VAR
	Document	  : SJsonValue;
	JsonAttribute : T_MaxString;
	TaskName	  : T_MaxString;
	temp		  : UDINT;
END_VAR

VAR_INST
	LastScanCount		 : UDINT;
	MessagesSentThisScan : UDINT;
	MissedMessages		 : UDINT;
	Throttled			 : BOOL;
END_VAR

VAR
	ThrottledNotificationString : T_MaxString;
	CurrentDCTime				: DCTIMESTRUCT;
	DCTime100Nsec				: WORD;
	DCTimeString				: T_MaxString;
END_VAR
IF NOT InitComplete THEN
	RETURN;
END_IF

{analysis -62}
IF NOT TracingAllowed THEN
	RETURN;
END_IF

IF NOT Parameters_Tracing.ALLOW_DUPLICATE_SEQUENTIAL_MESSAGES THEN
	IF (MEMCMP(ADR(Source), ADR(Previous_AddEntryJsonSource), SIZEOF(T_MaxString)) = 0) AND (MEMCMP(ADR(Message), ADR(Previous_AddEntryJsonMessage), SIZEOF(T_MaxString)) = 0) AND (Flags = Previous_AddEntryJsonFlags) AND (MEMCMP(ADR(Json), ADR(Previous_AddEntryJson), SIZEOF(T_MaxString)) = 0) THEN
		// This message is identical to the last message sent--ignore
		RETURN;
	END_IF
END_IF

Event.ipArguments.Clear().AddString(Message);
AddContext(Source := Source, Flags := Flags);
Document := JsonParser.NewDocument();
JsonParser.AddJsonMember(Document, 'ExtendedInfo', Json);
JsonAttribute := JsonParser.GetJson(Document);
Event.SetJsonAttribute(JsonAttribute);
Event.Send(0);
MessagesSentThisScan := MessagesSentThisScan + 1;
MEMCPY(ADR(Previous_AddEntryJsonSource), ADR(Source), SIZEOF(T_MaxString));
MEMCPY(ADR(Previous_AddEntryJsonMessage), ADR(Message), SIZEOF(T_MaxString));
Previous_AddEntryFlags := Flags;
MEMCPY(ADR(Previous_AddEntryJsonMessage), ADR(Json), SIZEOF(T_MaxString));
END_METHOD

METHOD FB_init : BOOL
VAR_INPUT
	bInitRetains : BOOL; // if TRUE, the retain variables are initialized (warm start / cold start)
	bInCopyCode	 : BOOL; // if TRUE, the instance afterwards gets moved into the copy code (online change)
END_VAR

VAR
	hr : HRESULT;
END_VAR
{analysis -15}
IF NOT Event.EqualsToEventEntryEx(TC_EVENTS.Tracing.TraceEvent) THEN
	IF SUCCEEDED(Event.CreateEx(TC_EVENTS.Tracing.TraceEvent, 0)) THEN
		InitComplete := TRUE;
	END_IF
ELSE
	InitComplete := TRUE;
END_IF
END_METHOD

PROPERTY PRIVATE TracingAllowed : BOOL
GET
VAR_INST
	LastScanCount  : UDINT;
	MissedMessages : UDINT;
	Throttled	   : BOOL;
END_VAR

VAR
	ThrottledNotificationString : T_MaxString;
END_VAR
{analysis -62}
IF NOT Parameters_Tracing.TRACING_ENABLED THEN
	TracingAllowed := FALSE;
	RETURN;
END_IF

IF TwinCAT_SystemInfoVarList._TaskInfo[GETCURTASKINDEXEX()].CycleCount = LastScanCount THEN
	// Trying to send multiple messages in same scan
	IF Throttled THEN
		MissedMessages := MissedMessages + 1;
		RETURN;
	ELSIF MessagesSentThisScan >= Parameters_Tracing.MAX_LOG_ENTRIES_PER_SCAN AND NOT Throttled THEN
		// Need to throttle messsage queue
		Event.ipArguments.Clear().AddString('Too many messages sent in single scan; tracing throttled.');
		Event.Send(0);
		MissedMessages := MissedMessages + 1;
		Throttled	   := TRUE;
		TracingAllowed := FALSE;
		RETURN;
	ELSE
		TracingAllowed := TRUE;
	END_IF
ELSE
	IF Throttled THEN
		ThrottledNotificationString := CONCAT('Missed ', CONCAT(TO_STRING(MissedMessages), ' throttled messages previously.'));
		Event.ipArguments.Clear().AddString(ThrottledNotificationString);
		Event.Send(0);
		MissedMessages := 0;
	END_IF

	LastScanCount		 := TwinCAT_SystemInfoVarList._TaskInfo[GETCURTASKINDEXEX()].CycleCount;
	MessagesSentThisScan := 0;
	Throttled			 := FALSE;
	TracingAllowed		 := TRUE;
END_IF
END_GET
END_PROPERTY

END_FUNCTION_BLOCK

// VISUs/V_MachineModule
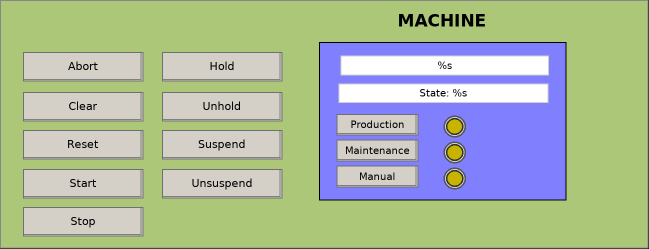
VISUALIZATION V_MachineModule  // 649x249
VAR_IN_OUT
	HMI : ST_PackMLBaseModule_HMI;
END_VAR
    RoundedRectangle (0,0 649x249)
    Button (23,52 120x29), "Abort"
        OnMouseClick: execute { HMI.Command.State := E_PMLCommand.ePMLCommand_Abort; }
    Button (23,92 120x29), "Clear"
        OnMouseClick: execute { HMI.Command.State := E_PMLCommand.ePMLCommand_Clear; }
    Button (23,130 120x29), "Reset"
        OnMouseClick: execute { HMI.Command.State := E_PMLCommand.ePMLCommand_Reset; }
    Button (23,169 120x29), "Start"
        OnMouseClick: execute { HMI.Command.State := E_PMLCommand.ePMLCommand_Start; }
    Button (23,207 120x29), "Stop"
        OnMouseClick: execute { HMI.Command.State := E_PMLCommand.ePMLCommand_Stop; }
    Button (162,52 120x29), "Hold"
        OnMouseClick: execute { HMI.Command.State := E_PMLCommand.ePMLCommand_Hold; }
    Button (162,92 120x29), "Unhold"
        OnMouseClick: execute { HMI.Command.State := E_PMLCommand.ePMLCommand_Unhold; }
    Button (162,130 120x29), "Suspend"
        OnMouseClick: execute { HMI.Command.State := E_PMLCommand.ePMLCommand_Suspend; }
    Button (162,169 120x29), "Unsuspend"
        OnMouseClick: execute { HMI.Command.State := E_PMLCommand.ePMLCommand_Unsuspend; }
    Frame (319,42 247x158)
        shows V_Module(HMI := HMI)
    Label (357,2 170x37), "MACHINE"
END_VISUALIZATION

// VISUs/V_Module
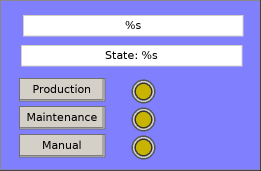
VISUALIZATION V_Module  // 261x171
VAR_IN_OUT
	HMI : ST_PackMLBaseModule_HMI;
END_VAR
    RoundedRectangle (0,0 261x171)
    Textfield (23,15 220x21), "%s", text variable: HMI.Config.Name
    Textfield (21,45 221x21), "State: %s", text variable: HMI.Status.State
    Button (19,78 86x23), "Production"
        OnMouseClick: execute { HMI.Command.Mode := E_PMLUnitMode.ePMLUnitMode_Production; }
    Button (19,106 86x23), "Maintenance"
        OnMouseClick: execute { HMI.Command.Mode := E_PMLUnitMode.ePMLUnitMode_Maintenance; }
    Button (19,134 86x23), "Manual"
        OnMouseClick: execute { HMI.Command.Mode := E_PMLUnitMode.ePMLUnitMode_Manual; }
    Lamp1 (130,78 27x27), variable: HMI.Status.Mode = E_PMLUnitMode.ePMLUnitMode_Production, style: Lamp-Lamp1-Yellow
    Lamp1 (130,106 27x27), variable: HMI.Status.Mode = E_PMLUnitMode.ePMLUnitMode_Maintenance, style: Lamp-Lamp1-Yellow
    Lamp1 (130,134 27x27), variable: HMI.Status.Mode = E_PMLUnitMode.ePMLUnitMode_Manual, style: Lamp-Lamp1-Yellow
END_VISUALIZATION
